{attribute 'qualified_only'}
{attribute 'strict'}
TYPE State :
(
	None,
	Stopped,
	Starting,
	Running,
	Pausing,
	Paused,
	Resuming,
	Stopping,
	Aborting,
	Aborted,
	Resetting	
);
END_TYPE

(* stored: Version 1.1.0.1, ProductVersion 3.1.4022.11
   DUT State: Id {711acabc-880c-4edb-97f9-25be82c11d70} *)
